FUNCTION_BLOCK INTERNAL FINAL FB_ReadRepeatedFieldFixed32Tests EXTENDS FB_TestSuite
VAR_INPUT
END_VAR
VAR_OUTPUT
END_VAR
VAR
	aActual             : ARRAY [0..7] OF DINT;
	fbFieldCodec 		: FB_FieldCodecFixed32(nTag:= 16#0A);
	fbRepeatedField	: FB_RepeatedField(anyArray:= F_ToAnyType(aActual), anyFirstElem:= F_ToAnyType(aActual[0]), ipFieldCodec:= fbFieldCodec);
END_VAR

ShouldReadRepeatedFieldTheory();

METHOD PRIVATE Reset
VAR_INPUT
END_VAR
fbRepeatedField.Initialize();
MEMSET(destAddr:= ADR(aActual), fillByte:= 16#0, n:= SIZEOF(aActual[0]));
END_METHOD

METHOD PRIVATE ShouldReadRepeatedField
VAR_IN_OUT CONSTANT
    aBuffer     : ARRAY [*] OF BYTE;
    aExpected   : ARRAY [*] OF DINT;
END_VAR
VAR_INPUT CONSTANT
    nBufferPosStart     : UDINT;
    nExpectedBufferPos  : UDINT;
    nExpectedFieldIndex : UDINT;
    ipFieldCodec        : I_FieldCodec;
END_VAR
VAR_INST
    fbCtx               : FB_ParseContext;
END_VAR
VAR
    hr                  : HRESULT;
	nTag                : UDINT;
END_VAR
// Arrange
Reset();
fbCtx.FromBuffer(aBuffer);
fbCtx.refCtx.stState.nBufferPos := nBufferPosStart;;

// Act
F_ParseTag(fbCtx.refCtx, nTag=> nTag);
hr := fbRepeatedField.AddEntriesFrom(fbParseCtx:= fbCtx, ipFieldCodec:= ipFieldCodec);

// Assert
AssertEquals_DINT(
    Expected:= S_OK,
    Actual:= hr,
    Message:= 'Expected S_OK instead of error');
    
{warning disable C0041}
AssertArrayEquals_DINT(Expecteds:= aExpected, Actuals:= aActual, Message:= '');
 
AssertEquals_UDINT(
    Expected:= nExpectedBufferPos,
    Actual:= fbCtx.refCtx.stState.nBufferPos,
    Message:= CONCAT('Expected stState.nBufferPos to equal ', TO_STRING(nExpectedBufferPos)));
    
AssertEquals_UDINT(
    Expected:= nExpectedFieldIndex,
    Actual:= fbRepeatedField.nCount,
    Message:= CONCAT('Expected fbRepeatedField.nCount to equal ', TO_STRING(nExpectedFieldIndex)));
END_METHOD

METHOD PRIVATE ShouldReadRepeatedFieldTheory : REFERENCE TO FB_Test
(*
    syntax = "proto3";
    
    message exampleMessage
    {
      repeated fixed32 repeatedFixed32 = 4;
    }
*)
VAR CONSTANT
    cRawValueZeroLength     : ARRAY[0..31] OF BYTE := [16#22, 16#00];       // field #4
    cRawValue1              : ARRAY[0..31] OF BYTE := [16#00, 16#22, 16#18, 16#00, 16#00, 16#00, 16#00, 16#D2, 16#04, 16#00, 16#00, 16#39, 16#05, 16#00, 16#00, 16#FF, 16#FF, 16#FF, 16#FF, 16#C7, 16#FA, 16#FF, 16#FF, 16#4E, 16#61, 16#BC, 16#00];
    
END_VAR

VAR CONSTANT
    aExpectedZeroLength     : ARRAY [0..7] OF DINT := [0, 0, 0, 0, 0, 0, 0, 0];
    aExpected1              : ARRAY [0..7] OF DINT := [0, 1234, 1337, -1, -1337, 12345678, 0, 0];
END_VAR
TEST(__POUNAME());

ShouldReadRepeatedField(aBuffer:= cRawValueZeroLength, aExpected:= aExpectedZeroLength, nBufferPosStart:= 0, nExpectedBufferPos:= 2, nExpectedFieldIndex:= 0, ipFieldCodec:= THIS^.fbFieldCodec);
ShouldReadRepeatedField(aBuffer:= cRawValue1, aExpected:= aExpected1, nBufferPosStart:= 1, nExpectedBufferPos:= 27, nExpectedFieldIndex:= 6, ipFieldCodec:= THIS^.fbFieldCodec);

TEST_FINISHED_NAMED(__POUNAME());
END_METHOD

END_FUNCTION_BLOCK

(* stored: Version 1.1.0.1
   POU FB_ReadRepeatedFieldFixed32Tests: Id {0262274a-c960-4ad8-92d1-7a52fe0fc4cd}, SpecialFunc None
   Method Reset: Id {a33328b2-d872-446d-93d0-07d1d546219b}
   Method ShouldReadRepeatedField: Id {f5e4b169-ab63-40a0-aad4-6ff8c1081522}
   Method ShouldReadRepeatedFieldTheory: Id {901da591-6ef9-463e-abbc-5aea1eb7096d} *)
